PROGRAM PRG_TEST
VAR
	fbDynamicMatrix : FB_DynamicMatrix_Test;
	fbMatrixGetMagicSquare : FB_MatrixGetMagicSquare_Test;
	fbMatrixSubmatrix : FB_MatrixSubMatrix_Test;
	fbMatrixGrow : FB_MatrixGrow_Test;
	fbMatrixShrink : FB_MatrixShrink_Test;
	fbMatrixElementSum : FB_MatrixElementSum_Test;
	fbMatrixElementProduct : FB_MatrixElementProduct_Test;
	fbMatrixDeterminate : FB_MatrixDeterminate_Test;
	fbMatrixMatrixProduct : FB_MatrixMatrixProduct_Test;
	fbVectorCrossProdcut : FB_VectorCrossProduct_Test;
	fbStaticMatrix : FB_StaticMatrix_Test;
	fbMatrixTranspose : FB_MatrixTranspose_Test;
	fbMatrixInvert : FB_MatrixInvert_Test;
END_VAR

TcUnit.RUN();

END_PROGRAM

(* stored: Version 1.1.0.1, ProductVersion 3.1.4024.9
   POU PRG_TEST: Id {5f2716c6-31ed-49cd-815d-6106c2eebb72}, SpecialFunc None *)
